# EPICS substitutions: viocs/substitutions/cvs.substitutions
file "db/individual.db" {
    pattern { family, pos }
        { "CVS", "01C1" }
        { "CVS", "01C2" }
        { "CVS", "01C3" }
        { "CVS", "01C4" }
        { "CVS", "01M1" }
        { "CVS", "01M2" }
        { "CVS", "02C1" }
        { "CVS", "02C2" }
        { "CVS", "02C3" }
        { "CVS", "02C4" }
        { "CVS", "02M1" }
        { "CVS", "02M2" }
        { "CVS", "03C1" }
        { "CVS", "03C2" }
        { "CVS", "03C3" }
        { "CVS", "03C4" }
        { "CVS", "03M1" }
        { "CVS", "03M2" }
        { "CVS", "04C1" }
        { "CVS", "04C2" }
        { "CVS", "04C3" }
        { "CVS", "04C4" }
        { "CVS", "04M1" }
        { "CVS", "04M2" }
        { "CVS", "05C1" }
        { "CVS", "05C2" }
        { "CVS", "05C3" }
        { "CVS", "05C4" }
        { "CVS", "05M1" }
        { "CVS", "05M2" }
        { "CVS", "06C1" }
        { "CVS", "06C2" }
        { "CVS", "06C3" }
        { "CVS", "06C4" }
        { "CVS", "06M1" }
        { "CVS", "06M2" }
        { "CVS", "07C1" }
        { "CVS", "07C2" }
        { "CVS", "07C3" }
        { "CVS", "07C4" }
        { "CVS", "07M1" }
        { "CVS", "07M2" }
        { "CVS", "08C1" }
        { "CVS", "08C2" }
        { "CVS", "08C3" }
        { "CVS", "08C4" }
        { "CVS", "08M1" }
        { "CVS", "08M2" }
        { "CVS", "09C1" }
        { "CVS", "09C2" }
        { "CVS", "09C3" }
        { "CVS", "09C4" }
        { "CVS", "09M1" }
        { "CVS", "09M2" }
        { "CVS", "10C1" }
        { "CVS", "10C2" }
        { "CVS", "10C3" }
        { "CVS", "10C4" }
        { "CVS", "10M1" }
        { "CVS", "10M2" }
        { "CVS", "11C1" }
        { "CVS", "11C2" }
        { "CVS", "11C3" }
        { "CVS", "11C4" }
        { "CVS", "11M1" }
        { "CVS", "11M2" }
        { "CVS", "12C1" }
        { "CVS", "12C2" }
        { "CVS", "12C3" }
        { "CVS", "12C4" }
        { "CVS", "12M1" }
        { "CVS", "12M2" }
        { "CVS", "13C1" }
        { "CVS", "13C2" }
        { "CVS", "13C3" }
        { "CVS", "13C4" }
        { "CVS", "13M1" }
        { "CVS", "13M2" }
        { "CVS", "14C1" }
        { "CVS", "14C2" }
        { "CVS", "14C3" }
        { "CVS", "14C4" }
        { "CVS", "14M1" }
        { "CVS", "14M2" }
        { "CVS", "15C1" }
        { "CVS", "15C2" }
        { "CVS", "15C3" }
        { "CVS", "15C4" }
        { "CVS", "15M1" }
        { "CVS", "15M2" }
        { "CVS", "16C1" }
        { "CVS", "16C2" }
        { "CVS", "16C3" }
        { "CVS", "16C4" }
        { "CVS", "16M1" }
        { "CVS", "16M2" }
        { "CVS", "17C1" }
        { "CVS", "17C2" }
        { "CVS", "17C3" }
        { "CVS", "17C4" }
        { "CVS", "17M1" }
        { "CVS", "17M2" }
        { "CVS", "18C1" }
        { "CVS", "18C2" }
        { "CVS", "18C3" }
        { "CVS", "18C4" }
        { "CVS", "18M1" }
        { "CVS", "18M2" }
        { "CVS", "19C1" }
        { "CVS", "19C2" }
        { "CVS", "19C3" }
        { "CVS", "19C4" }
        { "CVS", "19M1" }
        { "CVS", "19M2" }
        { "CVS", "20C1" }
        { "CVS", "20C2" }
        { "CVS", "20C3" }
        { "CVS", "20C4" }
        { "CVS", "20M1" }
        { "CVS", "20M2" }
}
